(*~
    <docu>
        <summary>
            Base block for interactive dialogs.
         </summary>
    </docu>
~*)
FUNCTION_BLOCK ABSTRACT TcoDialogBase EXTENDS TcoRemoteTask

SUPER^();

{attribute 'hide'}
METHOD PUBLIC FB_init : BOOL
VAR_INPUT
    bInitRetains : BOOL; // if TRUE, the retain variables are initialized (warm start / cold start)
    bInCopyCode : BOOL; // if TRUE, the instance afterwards gets moved into the copy code (online change)
    ParentObject : ITcoObject;
END_VAR
END_METHOD

METHOD PROTECTED OnStart
SUPER^.OnStart();
END_METHOD

END_FUNCTION_BLOCK

(* stored: Version 1.1.0.1
   POU TcoDialogBase: Id {b361351b-637d-0485-12e4-25b8c4bb42be}, SpecialFunc None
   Method FB_init: Id {8d8e4207-be67-0434-27e5-b762ade88dae}
   Method OnStart: Id {05c1ce12-e48b-0c1d-3ab0-55659aef6070} *)
